(* CODESYS project boiler2.project
   Title: testPrj
   Version: 0.0.0.0

Project tree, tasks and I/O mapping:
  MyController : TM241CE40R, Schneider Electric, order no. TM241CE40R, version 4.0.2.20
    application Application
      libraries: Toolbox, 2.1.0.0 (Schneider Electric); Util, 3.5.1.0 (System)
      task MAST (freewheeling, priority 15, watchdog 100 ms x 1) calls main, pid_control, XT_output
      task Dempf (cyclic, interval t#50ms, priority 1) calls Analog
      function HiddenPOU [ST]
      global variables GVL
      Prog/
        program main [ST]
        program Analog [FBD]
        program pid_control [FBD]
        program XT_output [ST]
        program SafeTmr [FBD]
    DI : Digital Inputs, Schneider Electric, version 4.0.2.20
        input  idwDI_IDW0 : DWORD  // IDW0
        input  Application.xDrumLH1 : BOOL  // IDW0.I0
        input  Application.xDrumLH2 : BOOL  // IDW0.I1
        input  Application.xDrumLl1 : BOOL  // IDW0.I2
        input  Application.xDrumLl2 : BOOL  // IDW0.I3
        input  Application.xFanRun : BOOL  // IDW0.I4
        input  Application.xExhRun : BOOL  // IDW0.I5
        input  Application.xPumpRun : BOOL  // IDW0.I6
        input  Application.xSafeOn : BOOL  // IDW0.I7
        input  Application.xDrumPh : BOOL  // IDW0.I8
        input  Application.xGasPl : BOOL  // IDW0.I9
        input  Application.xGasPh : BOOL  // IDW0.I10
        input  Application.xAirPl : BOOL  // IDW0.I11
        input  Application.xVacPl : BOOL  // IDW0.I12
        input  Application.xBump : BOOL  // IDW0.I13
        input  Application.xFire1 : BOOL  // IDW0.I14
        input  Application.xTight : BOOL  // IDW0.I15
        input  Application.xStartBn : BOOL  // IDW0.I16
        input  Application.xStopBn : BOOL  // IDW0.I17
        input  Application.xAlarmBn : BOOL  // IDW0.I18
        input  Application.xGasAuto : BOOL  // IDW0.I19
        input  Application.xTermAuto : BOOL  // IDW0.I20
        input  Application.xPumpAuto : BOOL  // IDW0.I21
        input  Application.xExhAuto : BOOL  // IDW0.I22
        input  Application.xFanAuto : BOOL  // IDW0.I23
        input  ibDI_IB1 : BYTE  // IB1
    DQ : Digital Outputs, Schneider Electric, version 4.0.2.20
        output Application.yTermOpen : BOOL  // QW0.Q0
        output Application.yTermClose : BOOL  // QW0.Q1
        output Application.ySuppOpen : BOOL  // QW0.Q2
        output Application.ySuppClose : BOOL  // QW0.Q3
        output Application.yCutofVal : BOOL  // QW0.Q4
        output Application.yBurnerVal : BOOL  // QW0.Q5
        output Application.ySafeVal : BOOL  // QW0.Q6
        output Application.yLitherVal : BOOL  // QW0.Q7
        output Application.yFanStart : BOOL  // QW0.Q8
        output Application.yPumpStart : BOOL  // QW0.Q9
        output Application.yGasOpen : BOOL  // QW0.Q10
        output Application.yGasClose : BOOL  // QW0.Q11
        output Application.yPlcStop : BOOL  // QW0.Q12
        output Application.ySerena : BOOL  // QW0.Q13
        output Application.yLamp : BOOL  // QW0.Q14
        output Application.yIgniter : BOOL  // QW0.Q15
        output qbDQ_QB1 : BYTE  // QB1
        unmapped channels: QW0
    Counters : Counters, Schneider Electric, version 4.0.2.20
    Pulse_Generators : Pulse Generators, Schneider Electric, version 4.0.2.20
    Cartridge_1 : Cartridge, Schneider Electric, version 4.0.2.20
    Cartridge_2 : Cartridge, Schneider Electric, version 4.0.2.20
    IO_Bus : IO bus - TM3, Schneider Electric, version 4.0.2.20
      Module_1 : TM3AQ4/G, Schneider Electric, order no. TM3AQ4/G, version 1.0.0.10
          settings: KPI Configuration.KPI Configuration[0] = 19; KPI Configuration.KPI Configuration[1] = 19; KPI Configuration.KPI Configuration[2] = 19; KPI Configuration.KPI Configuration[3] = 19; KPI Configuration.KPI Configuration[5] = 0; KPI Configuration.KPI Configuration[7] = 0; KPI Configuration.KPI Configuration[9] = 0; KPI Configuration.KPI Configuration[11] = 0; KPI Configuration.KPI Configuration[12] = 160; KPI Configuration.KPI Configuration[13] = 15; KPI Configuration.KPI Configuration[14] = 160; KPI Configuration.KPI Configuration[15] = 15; KPI Configuration.KPI Configuration[16] = 160; KPI Configuration.KPI Configuration[17] = 15; KPI Configuration.KPI Configuration[18] = 160; KPI Configuration.KPI Configuration[19] = 15
          output C0001 : INT  // QW0
          output C0002 : INT  // QW1
          output C0003 : INT  // QW2
          output C0004 : INT  // QW3
          input  ibModule_1_IBStatusQW0 : BYTE  // IBStatusQW0
          input  ibModule_1_IBStatusQW1 : BYTE  // IBStatusQW1
          input  ibModule_1_IBStatusQW2 : BYTE  // IBStatusQW2
          input  ibModule_1_IBStatusQW3 : BYTE  // IBStatusQW3
      Module_2 : TM3AI8/G, Schneider Electric, order no. TM3AI8/G, version 1.0.0.12
          settings: KPI Configuration.KPI Configuration[0] = 35; KPI Configuration.KPI Configuration[1] = 35; KPI Configuration.KPI Configuration[2] = 35; KPI Configuration.KPI Configuration[3] = 35; KPI Configuration.KPI Configuration[4] = 35; KPI Configuration.KPI Configuration[5] = 35; KPI Configuration.KPI Configuration[6] = 35; KPI Configuration.KPI Configuration[7] = 35; KPI Configuration.KPI Configuration[9] = 0; KPI Configuration.KPI Configuration[11] = 0; KPI Configuration.KPI Configuration[13] = 0; KPI Configuration.KPI Configuration[15] = 0; KPI Configuration.KPI Configuration[17] = 0; KPI Configuration.KPI Configuration[19] = 0; KPI Configuration.KPI Configuration[21] = 0; KPI Configuration.KPI Configuration[23] = 0; KPI Configuration.KPI Configuration[24] = 160; KPI Configuration.KPI Configuration[25] = 15; KPI Configuration.KPI Configuration[26] = 160; KPI Configuration.KPI Configuration[27] = 15; KPI Configuration.KPI Configuration[28] = 160; KPI Configuration.KPI Configuration[29] = 15; KPI Configuration.KPI Configuration[30] = 160; KPI Configuration.KPI Configuration[31] = 15; KPI Configuration.KPI Configuration[32] = 160; KPI Configuration.KPI Configuration[33] = 15; KPI Configuration.KPI Configuration[34] = 160; KPI Configuration.KPI Configuration[35] = 15; KPI Configuration.KPI Configuration[36] = 160; KPI Configuration.KPI Configuration[37] = 15; KPI Configuration.KPI Configuration[38] = 160; KPI Configuration.KPI Configuration[39] = 15
          input  A0000 : INT  // IW0
          input  A0001 : INT  // IW1
          input  A0002 : INT  // IW2
          input  A0003 : INT  // IW3
          input  A0004 : INT  // IW4
          input  A0005 : INT  // IW5
          input  A0006 : INT  // IW6
          input  A0007 : INT  // IW7
          input  ibModule_2_IBStatusIW0 : BYTE  // IBStatusIW0
          input  ibModule_2_IBStatusIW1 : BYTE  // IBStatusIW1
          input  ibModule_2_IBStatusIW2 : BYTE  // IBStatusIW2
          input  ibModule_2_IBStatusIW3 : BYTE  // IBStatusIW3
          input  ibModule_2_IBStatusIW4 : BYTE  // IBStatusIW4
          input  ibModule_2_IBStatusIW5 : BYTE  // IBStatusIW5
          input  ibModule_2_IBStatusIW6 : BYTE  // IBStatusIW6
          input  ibModule_2_IBStatusIW7 : BYTE  // IBStatusIW7
      Module_3 : TM3AI8/G, Schneider Electric, order no. TM3AI8/G, version 1.0.0.12
          settings: KPI Configuration.KPI Configuration[0] = 35; KPI Configuration.KPI Configuration[1] = 35; KPI Configuration.KPI Configuration[2] = 35; KPI Configuration.KPI Configuration[3] = 35; KPI Configuration.KPI Configuration[4] = 35; KPI Configuration.KPI Configuration[5] = 35; KPI Configuration.KPI Configuration[6] = 35; KPI Configuration.KPI Configuration[7] = 35; KPI Configuration.KPI Configuration[9] = 0; KPI Configuration.KPI Configuration[11] = 0; KPI Configuration.KPI Configuration[13] = 0; KPI Configuration.KPI Configuration[15] = 0; KPI Configuration.KPI Configuration[17] = 0; KPI Configuration.KPI Configuration[19] = 0; KPI Configuration.KPI Configuration[21] = 0; KPI Configuration.KPI Configuration[23] = 0; KPI Configuration.KPI Configuration[24] = 160; KPI Configuration.KPI Configuration[25] = 15; KPI Configuration.KPI Configuration[26] = 160; KPI Configuration.KPI Configuration[27] = 15; KPI Configuration.KPI Configuration[28] = 160; KPI Configuration.KPI Configuration[29] = 15; KPI Configuration.KPI Configuration[30] = 160; KPI Configuration.KPI Configuration[31] = 15; KPI Configuration.KPI Configuration[32] = 160; KPI Configuration.KPI Configuration[33] = 15; KPI Configuration.KPI Configuration[34] = 160; KPI Configuration.KPI Configuration[35] = 15; KPI Configuration.KPI Configuration[36] = 232; KPI Configuration.KPI Configuration[37] = 3; KPI Configuration.KPI Configuration[38] = 160; KPI Configuration.KPI Configuration[39] = 15
          input  A0010 : INT  // IW0
          input  A0011 : INT  // IW1
          input  A0012 : INT  // IW2
          input  A0013 : INT  // IW3
          input  A0014 : INT  // IW4
          input  A0015 : INT  // IW5
          input  A0016 : INT  // IW6
          input  A0017 : INT  // IW7
          input  ibModule_3_IBStatusIW0 : BYTE  // IBStatusIW0
          input  ibModule_3_IBStatusIW1 : BYTE  // IBStatusIW1
          input  ibModule_3_IBStatusIW2 : BYTE  // IBStatusIW2
          input  ibModule_3_IBStatusIW3 : BYTE  // IBStatusIW3
          input  ibModule_3_IBStatusIW4 : BYTE  // IBStatusIW4
          input  ibModule_3_IBStatusIW5 : BYTE  // IBStatusIW5
          input  ibModule_3_IBStatusIW6 : BYTE  // IBStatusIW6
          input  ibModule_3_IBStatusIW7 : BYTE  // IBStatusIW7
      Module_4 : TM3AI8/G, Schneider Electric, order no. TM3AI8/G, version 1.0.0.12
          settings: KPI Configuration.KPI Configuration[0] = 35; KPI Configuration.KPI Configuration[1] = 35; KPI Configuration.KPI Configuration[2] = 35; KPI Configuration.KPI Configuration[3] = 35; KPI Configuration.KPI Configuration[4] = 35; KPI Configuration.KPI Configuration[5] = 35; KPI Configuration.KPI Configuration[6] = 35; KPI Configuration.KPI Configuration[7] = 35; KPI Configuration.KPI Configuration[9] = 0; KPI Configuration.KPI Configuration[11] = 0; KPI Configuration.KPI Configuration[13] = 0; KPI Configuration.KPI Configuration[15] = 0; KPI Configuration.KPI Configuration[17] = 0; KPI Configuration.KPI Configuration[19] = 0; KPI Configuration.KPI Configuration[21] = 0; KPI Configuration.KPI Configuration[23] = 0; KPI Configuration.KPI Configuration[24] = 160; KPI Configuration.KPI Configuration[25] = 15; KPI Configuration.KPI Configuration[26] = 160; KPI Configuration.KPI Configuration[27] = 15; KPI Configuration.KPI Configuration[28] = 160; KPI Configuration.KPI Configuration[29] = 15; KPI Configuration.KPI Configuration[30] = 160; KPI Configuration.KPI Configuration[31] = 15; KPI Configuration.KPI Configuration[32] = 160; KPI Configuration.KPI Configuration[33] = 15; KPI Configuration.KPI Configuration[34] = 160; KPI Configuration.KPI Configuration[35] = 15; KPI Configuration.KPI Configuration[36] = 160; KPI Configuration.KPI Configuration[37] = 15; KPI Configuration.KPI Configuration[38] = 160; KPI Configuration.KPI Configuration[39] = 15
          input  A0020 : INT  // IW0
          input  A0021 : INT  // IW1
          input  A0022 : INT  // IW2
          input  A0023 : INT  // IW3
          input  A0024 : INT  // IW4
          input  A0025 : INT  // IW5
          input  A0026 : INT  // IW6
          input  A0027 : INT  // IW7
          input  ibModule_4_IBStatusIW0 : BYTE  // IBStatusIW0
          input  ibModule_4_IBStatusIW1 : BYTE  // IBStatusIW1
          input  ibModule_4_IBStatusIW2 : BYTE  // IBStatusIW2
          input  ibModule_4_IBStatusIW3 : BYTE  // IBStatusIW3
          input  ibModule_4_IBStatusIW4 : BYTE  // IBStatusIW4
          input  ibModule_4_IBStatusIW5 : BYTE  // IBStatusIW5
          input  ibModule_4_IBStatusIW6 : BYTE  // IBStatusIW6
          input  ibModule_4_IBStatusIW7 : BYTE  // IBStatusIW7
    COM_Bus : COM bus, Schneider Electric, version 4.0.2.20
    Ethernet_1 : Ethernet Network, Schneider Electric, version 4.0.2.20
        settings: IPAddress = [192, 168, 15, 152]; SubnetMask = [255, 255, 255, 0]; GatewayAddress = [192, 168, 15, 1]; DeviceName = 'boiler2'; WebServer = FALSE; FTP Server = FALSE; SoMachine Protocol = TRUE; Modbus Server = TRUE; NetManage Protocol = FALSE; SNMP protocol = FALSE; Enable Routing = FALSE; WebVisu protocol = FALSE
      ModbusTCP_Slave_Device : ModbusTCP Slave Device, Schneider Electric, version 3.5.2.3
          unmapped channels: Inputs, Outputs
    Serial_Line_1 : Serial line, Schneider Electric, version 4.0.2.20
    Serial_Line_2 : Serial line, Schneider Electric, version 4.0.2.20
      Modbus_IOScanner : Modbus IOScanner, Schneider Electric, version 3.5.3.6
        Generic_Modbus_Slave : Generic Modbus Slave, Schneider Electric, version 3.5.3.6
            settings: Channel 1.Function Code = 3; Channel 1.Read Offset = 16#1001; Channel 1.Read Length = 6; Channel 1.Write Offset = 0; Channel 1.Write Length = 0; Channel 1.Cycle Time = 100; Channel 2.Function Code = 3; Channel 2.Read Offset = 16#8000; Channel 2.Read Length = 1; Channel 2.Write Offset = 0; Channel 2.Write Length = 0; Channel 2.Cycle Time = 100; Channel 3.Function Code = 3; Channel 3.Read Offset = 16#3000; Channel 3.Read Length = 1; Channel 3.Write Offset = 0; Channel 3.Write Length = 0; Channel 3.Cycle Time = 100
            input  M1 : WORD  // Channel 1.Channel 1[0]
            input  M2 : WORD  // Channel 1.Channel 1[1]
            input  M3 : WORD  // Channel 1.Channel 1[2]
            input  M4 : WORD  // Channel 1.Channel 1[3]
            input  M5 : WORD  // Channel 1.Channel 1[4]
            input  M6 : WORD  // Channel 1.Channel 1[5]
            input  M7 : WORD  // Channel 2.Channel 2[0]
            input  M8 : WORD  // Channel 3.Channel 3[0]
            unmapped channels: Channel 1, Channel 2, Channel 3
*)

// MyController/Application/GVL
VAR_GLOBAL

// run
	Run AT %M9: BOOL;
// DI
xDrumLH1 AT %M10: BOOL;
xDrumLH2 AT %M11: BOOL;
xDrumLl1 AT %M12: BOOL;
xDrumLl2 AT %M13: BOOL;
xFanRun AT %M14: BOOL;
xExhRun AT %M15: BOOL;
xPumpRun AT %M16: BOOL;
xSafeOn AT %M17: BOOL;
xDrumPh AT %M18: BOOL;
xGasPl AT %M19: BOOL;
xGasPh AT %M20: BOOL;
xAirPl AT %M21: BOOL;
xVacPl AT %M22: BOOL;
xBump AT %M23: BOOL;
xFire1 AT %M24: BOOL;
xTight AT %M25: BOOL;
xStartBn AT %M26: BOOL;
xStopBn AT %M27: BOOL;
xAlarmBn AT %M28: BOOL;
xGasAuto AT %M29: BOOL;
xTermAuto AT %M30: BOOL;
xPumpAuto AT %M31: BOOL;
xExhAuto AT %M32: BOOL;
xFanAuto AT %M33: BOOL;
// DO
yCutofVal AT %M34: BOOL;
yBurnerVal AT %M35: BOOL;
ySafeVal AT %M36: BOOL;
yLitherVal AT %M37: BOOL;
yIgniter AT %M38: BOOL;
yFanStart AT %M39: BOOL;
yPumpStart AT %M40: BOOL;
yGasOpen AT %M41: BOOL;
yGasClose AT %M42: BOOL;
yTermOpen AT %M43: BOOL;
yTermClose AT %M44: BOOL;
ySuppOpen AT %M45: BOOL;
ySuppClose AT %M46: BOOL;
yPlcStop AT %M47: BOOL;
ySerena AT %M48: BOOL;
yLamp AT %M49: BOOL;
//прапори аварійних сигналів
Alm0001 AT %M50: BOOL;
Alm0002 AT %M51: BOOL;
Alm0003 AT %M52: BOOL;
Alm0004 AT %M53: BOOL;
Alm0005 AT %M54: BOOL;
Alm0006 AT %M55: BOOL;
Alm0007 AT %M56: BOOL;
Alm0008 AT %M57: BOOL;
Alm0009 AT %M58: BOOL;
Alm0010 AT %M59: BOOL;
Alm0011 AT %M60: BOOL;
Alm0012 AT %M61: BOOL;
alFire1 AT %M62: BOOL;
alFan AT %M63: BOOL;
alExh AT %M64: BOOL;
alPump AT %M65: BOOL;
alSupport AT %M66: BOOL;

Alert AT %M123: BOOL;
Halt AT %M124: BOOL;
prLock AT %M125: BOOL;
Cvit AT %M126: BOOL;


amGas AT %M100: BOOL;
amTerm AT %M101: BOOL;
amSupport AT %M102: BOOL;
AM0001 AT %M103: BOOL;
AM0002 AT %M104: BOOL;
AM0003 AT %M105: BOOL;
AM0004 AT %M106: BOOL;
AM0005 AT %M107: BOOL;
AM0006 AT %M108: BOOL;



Fgas AT %MD9: REAL;
Fpara AT %MD10: REAL;
Fwater AT %MD11: REAL;
Fair AT %MD12: REAL;
Ldrum AT %MD13: REAL;
Pg15a AT %MD14: REAL;
Ppara AT %MD15: REAL;
Pp7a AT %MD16: REAL;

Tpar AT %MD17: REAL;
Tv3a AT %MD18: REAL;
Tv4a AT %MD19: REAL;
Tk AT %MD20: REAL;
Ta5a AT %MD21: REAL;
Ta6a AT %MD22: REAL;
Tp17a AT %MD23: REAL;
Tp18a AT %MD24: REAL;

Pair AT %MD25: REAL;
Pvac AT %MD26: REAL;
Pv12a AT %MD27: REAL;
gGas AT %MD28: REAL;
gTerm AT %MD49: REAL;
gSupp AT %MD51: REAL;
QO2fume AT %MD53: REAL;
Vx AT %MD55: REAL;

cPump AT %MD57: REAL;
cFan AT %MD59: REAL;
cExh AT %MD61: REAL;
cGas AT %MD63: REAL;
cTerm AT %MD65: REAL;
cSupport AT %MD67: REAL;
cX AT %MD69: REAL;


fA0000 AT %MW100: UINT;
fA0001 AT %MW101: UINT;
fA0002 AT %MW102: UINT;
fA0003 AT %MW103: UINT;
fA0004 AT %MW104: UINT;
fA0005 AT %MW105: UINT;
fA0006 AT %MW106: UINT;
fA0007 AT %MW107: UINT;
fA0010 AT %MW108: UINT;
fA0011 AT %MW109: UINT;
fA0012 AT %MW110: UINT;
fA0013 AT %MW111: UINT;
fA0014 AT %MW112: UINT;
fA0015 AT %MW113: UINT;
fA0016 AT %MW114: UINT;
fA0017 AT %MW115: UINT;
fA0020 AT %MW116: UINT;
fA0021 AT %MW117: UINT;
fA0022 AT %MW118: UINT;
fA0023 AT %MW119: UINT;
fA0024 AT %MW120: UINT;
fA0025 AT %MW121: UINT;
fA0026 AT %MW122: UINT;
fA0027 AT %MW123: UINT;

dGas AT %MD124: REAL;
dTerm AT %MD126: REAL;
dSupport AT %MD127: REAL;

Sp0001 AT %MD377: REAL;
Kp0001 AT %MD379: REAL;
Ti0001 AT %MD381: REAL;
Td0001 AT %MD383: REAL;
Xmin0001 AT %MD385: REAL;
Xmax0001 AT %MD387: REAL;

Sp0002 AT %MD389: REAL;
Kp0002 AT %MD391: REAL;
Ti0002 AT %MD393: REAL;
Td0002 AT %MD395: REAL;
Xmin0002 AT %MD397: REAL;
Xmax0002 AT %MD399: REAL;

Sp0003 AT %MD401: REAL;
Kp0003 AT %MD403: REAL;
Ti0003 AT %MD405: REAL;
Td0003 AT %MD407: REAL;
Xmin0003 AT %MD409: REAL;
Xmax0003 AT %MD411: REAL;

Sp0004 AT %MD413: REAL;
Kp0004 AT %MD415: REAL;
Ti0004 AT %MD417: REAL;
Td0004 AT %MD419: REAL;
Xmin0004 AT %MD421: REAL;
Xmax0004 AT %MD423: REAL;

Sp0005 AT %MD425: REAL;
Kp0005 AT %MD427: REAL;
Ti0005 AT %MD429: REAL;
Td0005 AT %MD431: REAL;
Xmin0005 AT %MD433: REAL;
Xmax0005 AT %MD435: REAL;

Sp0006 AT %MD437: REAL;
Kp0006 AT %MD439: REAL;
Ti0006 AT %MD441: REAL;
Td0006 AT %MD443: REAL;
Xmin0006 AT %MD445: REAL;
Xmax0006 AT %MD447: REAL;
// таймери аварій мео
tMeoTerm AT %MD449: REAL;
tMeoGas AT %MD451: REAL;

// таймери аварійних сигналізацій
Tpr0001 AT %ML511: TIME;
Tpr0002 AT %ML513: TIME;
Tpr0003 AT %ML515: TIME;
Tpr0004 AT %ML517: TIME;
Tpr0005 AT %ML519: TIME;
Tpr0006 AT %ML521: TIME;
Tpr0007 AT %ML523: TIME;
Tpr0008 AT %ML525: TIME;
Tpr0009 AT %ML527: TIME;
Tpr0010 AT %ML529: TIME;
Tpr0011 AT %ML531: TIME;
Tpr0012 AT %ML533: TIME;

	Xt0001: REAL;
	Xt0002: REAL;
	Xt0003: REAL;
	Xt0004: REAL;
	Xt0005: REAL;
	Xt0006: REAL;
	
	tMeo1: TIME;
	tMeo2: TIME;
	tMeo3: TIME;

END_VAR

// MyController/Application/Prog/main
PROGRAM main
VAR
	fe_amGas: F_TRIG;
	fe_amTerm: F_TRIG;
	fe_amSupport: F_TRIG;
END_VAR

(*Робота з МЕО*)
(*Газ*)
(*Взагалі-то вся ця хрінь проситься зробити блоком але як тоді в ручну управляти виходами ? треба подумати*)
IF amGas OR AM0004 THEN
	IF gGas>cGas+dGas THEN (*якщо відкрито більше ніж треба*)
		IF NOT yGasClose THEN (*В перший момент розрахувати значення таймера на виконання операції*) 
			tMeo1:=REAL_TO_TIME(ABS(gGas-cGas)*tMeoGas);
		END_IF;		
		yGasClose:=TRUE; (*відкрити*)
	END_IF;
	IF gGas<cGas-dGas THEN (*як закрито більше ніж треба*)
		IF NOT yGasOpen THEN 
			tMeo1:=REAL_TO_TIME(ABS(gGas-cGas)*tMeoGas);
		END_IF;		
		yGasOpen:=TRUE;
	END_IF;
	IF gGas<cGas THEN
		yGasClose:=FALSE;
	END_IF;
	IF gGas>cGas THEN 
		yGasOpen:=FALSE;
	END_IF;
END_IF;

(*при переході в ручний режим виключити виходи, якщов включені*)
fe_amGas(CLK:=amGas);
IF fe_amGas.Q THEN
	yGasOpen:=FALSE;
	yGasClose:=FALSE;
END_IF;


(*Температура*)
IF amTerm OR AM0005 THEN
	IF gTerm>cTerm+dTerm THEN (*якщо відкрито більге ніж треба*)
		IF NOT yTermClose THEN
			tMeo2:=REAL_TO_TIME(ABS(gTerm-cTerm)*tMeoTerm);		
		END_IF;
		yTermClose:=TRUE; (*відкрити*)
	END_IF;
	IF gTerm<cTerm-dTerm THEN (*як закрито більше ніж треба*)
		IF NOT yTermOpen THEN
			tMeo2:=REAL_TO_TIME(ABS(gTerm-cTerm)*tMeoTerm);		
		END_IF;
		tMeo2:=REAL_TO_TIME(ABS(gTerm-cTerm)*tMeoTerm);
		yTermOpen:=TRUE;
	END_IF;
	IF gTerm<cTerm THEN
		yTermClose:=FALSE;
	END_IF;
	IF gTerm>cTerm THEN 
		yTermOpen:=FALSE;
	END_IF;
END_IF;

(*при переході в ручний режим виключити виходи, якщов включені*)
fe_amTerm(CLK:=amTerm);
IF fe_amTerm.Q THEN
	yTermOpen:=FALSE;
	yTermClose:=FALSE;
END_IF;

(*підпір*)
IF amSupport OR AM0005  THEN
	cSupport:=4000.0-cTerm; (*клапан підпору працює в противофазі із клапаном температури*)
	IF gSupp>cSupport+dSupport THEN (*якщо відкрито більге ніж треба*)
		IF NOT ySuppClose THEN
			tMeo3:=REAL_TO_TIME(ABS(gSupp-cSupport)*tMeoTerm);				
		END_IF;
		ySuppClose:=TRUE; (*відкрити*)
	END_IF;
	IF gSupp<cSupport-dSupport THEN (*як закрито більше ніж треба*)
		IF NOT ySuppOpen THEN
			tMeo3:=REAL_TO_TIME(ABS(gSupp-cSupport)*tMeoTerm);		
		END_IF;
		ySuppOpen:=TRUE;
	END_IF;
	IF gSupp<cSupport THEN
		ySuppClose:=FALSE;
	END_IF;
	IF gSupp>cSupport THEN 
		ySuppOpen:=FALSE;
	END_IF;
END_IF;

(*при переході в ручний режим виключити виходи, якщов включені*)
fe_amSupport(CLK:=amSupport);
IF fe_amSupport.Q THEN
	ySuppOpen:=FALSE;
	ySuppClose:=FALSE;
END_IF;
(*----------------------------------------------------------------------------------------------------------------------------------*)

END_PROGRAM

// MyController/Application/Prog/pid_control
PROGRAM pid_control
VAR
	pid1: Util.PID;
	pid2: Util.PID;
	pid3: Util.PID;
	pid4: Util.PID;
	pid5: Util.PID;
	pid6: Util.PID;
END_VAR
VAR // added by the converter: edge detectors and wires of the graphical bodies
    _rt1, _rt2, _rt3, _rt4, _rt5, _rt6 : R_TRIG;
END_VAR

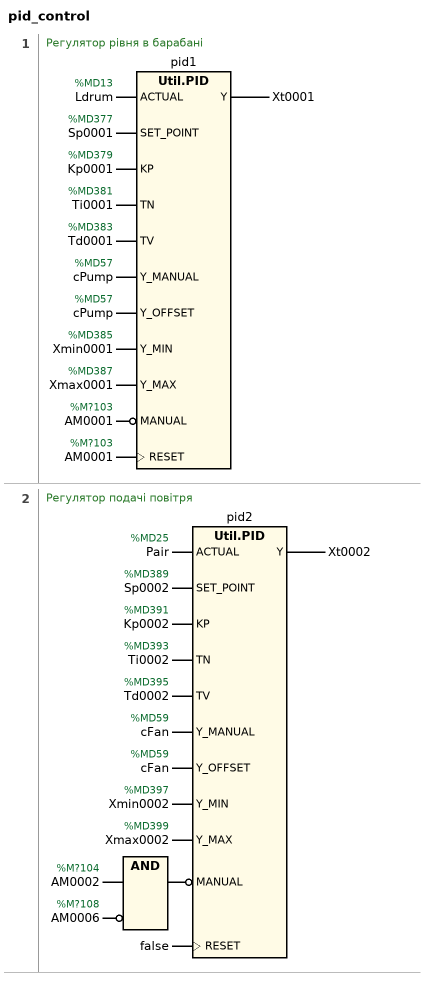
// NETWORK 1
// Регулятор рівня в барабані
//   Ldrum: AT %MD13
//   Sp0001: AT %MD377
//   Kp0001: AT %MD379
//   Ti0001: AT %MD381
//   Td0001: AT %MD383
//   cPump: AT %MD57
//   Xmin0001: AT %MD385
//   Xmax0001: AT %MD387
//   AM0001: AT %M?103
_rt1(CLK := AM0001);
pid1(
    ACTUAL := Ldrum,
    SET_POINT := Sp0001,
    KP := Kp0001,
    TN := Ti0001,
    TV := Td0001,
    Y_MANUAL := cPump,
    Y_OFFSET := cPump,
    Y_MIN := Xmin0001,
    Y_MAX := Xmax0001,
    MANUAL := NOT AM0001,
    RESET := _rt1.Q); // Util.PID
Xt0001 := pid1.Y;

// NETWORK 2
// Регулятор подачі повітря
//   Pair: AT %MD25
//   Sp0002: AT %MD389
//   Kp0002: AT %MD391
//   Ti0002: AT %MD393
//   Td0002: AT %MD395
//   cFan: AT %MD59
//   Xmin0002: AT %MD397
//   Xmax0002: AT %MD399
//   AM0002: AT %M?104
//   AM0006: AT %M?108
_rt2(CLK := false);
pid2(
    ACTUAL := Pair,
    SET_POINT := Sp0002,
    KP := Kp0002,
    TN := Ti0002,
    TV := Td0002,
    Y_MANUAL := cFan,
    Y_OFFSET := cFan,
    Y_MIN := Xmin0002,
    Y_MAX := Xmax0002,
    MANUAL := NOT (AM0002 AND NOT AM0006),
    RESET := _rt2.Q); // Util.PID
Xt0002 := pid2.Y;

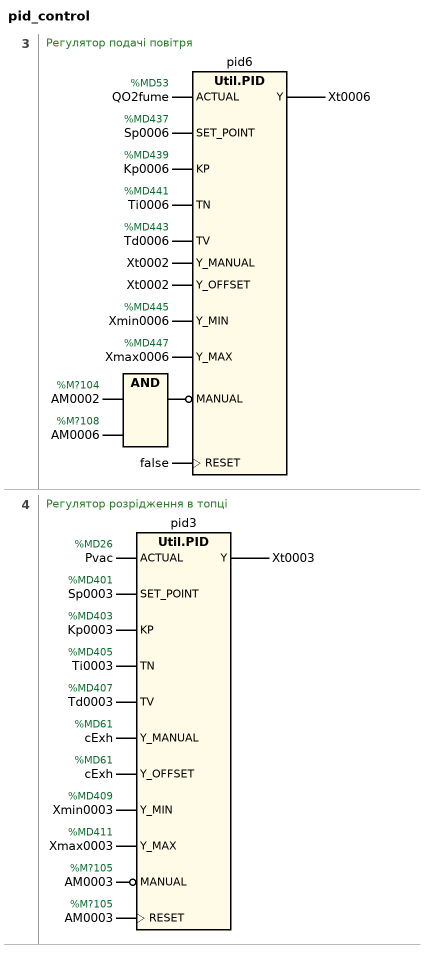
// NETWORK 3
// Регулятор подачі повітря
//   QO2fume: AT %MD53
//   Sp0006: AT %MD437
//   Kp0006: AT %MD439
//   Ti0006: AT %MD441
//   Td0006: AT %MD443
//   Xmin0006: AT %MD445
//   Xmax0006: AT %MD447
//   AM0002: AT %M?104
//   AM0006: AT %M?108
_rt3(CLK := false);
pid6(
    ACTUAL := QO2fume,
    SET_POINT := Sp0006,
    KP := Kp0006,
    TN := Ti0006,
    TV := Td0006,
    Y_MANUAL := Xt0002,
    Y_OFFSET := Xt0002,
    Y_MIN := Xmin0006,
    Y_MAX := Xmax0006,
    MANUAL := NOT (AM0002 AND AM0006),
    RESET := _rt3.Q); // Util.PID
Xt0006 := pid6.Y;

// NETWORK 4
// Регулятор розрідження в топці
//   Pvac: AT %MD26
//   Sp0003: AT %MD401
//   Kp0003: AT %MD403
//   Ti0003: AT %MD405
//   Td0003: AT %MD407
//   cExh: AT %MD61
//   Xmin0003: AT %MD409
//   Xmax0003: AT %MD411
//   AM0003: AT %M?105
_rt4(CLK := AM0003);
pid3(
    ACTUAL := Pvac,
    SET_POINT := Sp0003,
    KP := Kp0003,
    TN := Ti0003,
    TV := Td0003,
    Y_MANUAL := cExh,
    Y_OFFSET := cExh,
    Y_MIN := Xmin0003,
    Y_MAX := Xmax0003,
    MANUAL := NOT AM0003,
    RESET := _rt4.Q); // Util.PID
Xt0003 := pid3.Y;

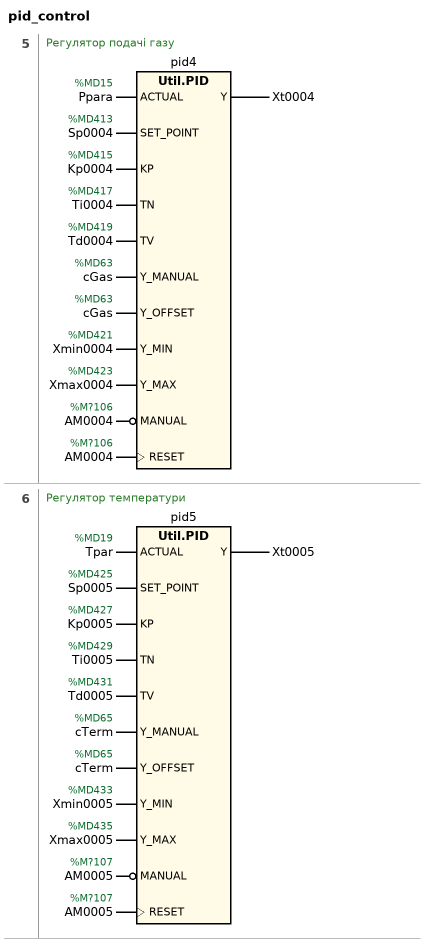
// NETWORK 5
// Регулятор подачі газу
//   Ppara: AT %MD15
//   Sp0004: AT %MD413
//   Kp0004: AT %MD415
//   Ti0004: AT %MD417
//   Td0004: AT %MD419
//   cGas: AT %MD63
//   Xmin0004: AT %MD421
//   Xmax0004: AT %MD423
//   AM0004: AT %M?106
_rt5(CLK := AM0004);
pid4(
    ACTUAL := Ppara,
    SET_POINT := Sp0004,
    KP := Kp0004,
    TN := Ti0004,
    TV := Td0004,
    Y_MANUAL := cGas,
    Y_OFFSET := cGas,
    Y_MIN := Xmin0004,
    Y_MAX := Xmax0004,
    MANUAL := NOT AM0004,
    RESET := _rt5.Q); // Util.PID
Xt0004 := pid4.Y;

// NETWORK 6
// Регулятор температури
//   Tpar: AT %MD19
//   Sp0005: AT %MD425
//   Kp0005: AT %MD427
//   Ti0005: AT %MD429
//   Td0005: AT %MD431
//   cTerm: AT %MD65
//   Xmin0005: AT %MD433
//   Xmax0005: AT %MD435
//   AM0005: AT %M?107
_rt6(CLK := AM0005);
pid5(
    ACTUAL := Tpar,
    SET_POINT := Sp0005,
    KP := Kp0005,
    TN := Ti0005,
    TV := Td0005,
    Y_MANUAL := cTerm,
    Y_OFFSET := cTerm,
    Y_MIN := Xmin0005,
    Y_MAX := Xmax0005,
    MANUAL := NOT AM0005,
    RESET := _rt6.Q); // Util.PID
Xt0005 := pid5.Y;

END_PROGRAM

// MyController/Application/Prog/XT_output
PROGRAM XT_output
VAR
	fe_am0001: F_TRIG;
	fe_am0002: F_TRIG;
	fe_am0003: F_TRIG;
	fe_am0004: F_TRIG;
	fe_am0005: F_TRIG;

	re_am0001: R_TRIG;
	re_am0002: R_TRIG;
	re_am0003: R_TRIG;
	re_am0004: R_TRIG;
	re_am0005: R_TRIG;

END_VAR

IF Am0001 THEN
	cPump:=Xt0001;
END_IF;

IF Am0002 THEN
	cFan:=Xt0006;
END_IF;

IF Am0003 THEN
	cExh:=Xt0003;
END_IF;

IF Am0004 THEN
	cGas:=Xt0004;
END_IF;

IF Am0005 THEN
	cTerm:=Xt0005;
END_IF;

(*Управління перемикачами ручний-автомати*)
re_AM0001(CLK:=xPumpAuto);
fe_AM0001(CLK:=xPumpAuto);

IF re_AM0001.Q THEN
	AM0001:=TRUE;
END_IF;

IF fe_AM0001.Q THEN
	AM0001:=FALSE;
END_IF;
(*-------------------------------------*)
re_AM0002(CLK:=xFanAuto);
fe_AM0002(CLK:=xFanAuto);

IF re_AM0002.Q THEN
	AM0002:=TRUE;
END_IF;

IF fe_AM0002.Q THEN
	AM0002:=FALSE;
END_IF;
(*-------------------------------------*)
re_AM0003(CLK:=xExhAuto);
fe_AM0003(CLK:=xExhAuto);

IF re_AM0003.Q THEN
	AM0003:=TRUE;
END_IF;

IF fe_AM0003.Q THEN
	AM0003:=FALSE;
END_IF;
(*-------------------------------------*)
re_AM0004(CLK:=xGasAuto);
fe_AM0004(CLK:=xGasAuto);

IF re_AM0004.Q THEN
	AM0004:=TRUE;
END_IF;

IF fe_AM0004.Q THEN
	AM0004:=FALSE;
END_IF;
(*-------------------------------------*)
re_AM0005(CLK:=xTermAuto);
fe_AM0005(CLK:=xTermAuto);

IF re_AM0005.Q THEN
	AM0005:=TRUE;
END_IF;

IF fe_AM0005.Q THEN
	AM0005:=FALSE;
END_IF;
(*-------------------------------------*)

END_PROGRAM

// MyController/Application/Prog/Analog
PROGRAM Analog
VAR
avg0000: SE_TBX.Filter_MovingAverage;
avg0001: SE_TBX.Filter_MovingAverage;
avg0002: SE_TBX.Filter_MovingAverage;
avg0003: SE_TBX.Filter_MovingAverage;
avg0004: SE_TBX.Filter_MovingAverage;
avg0005: SE_TBX.Filter_MovingAverage;
avg0006: SE_TBX.Filter_MovingAverage;
avg0007: SE_TBX.Filter_MovingAverage;
avg0010: SE_TBX.Filter_MovingAverage;
avg0011: SE_TBX.Filter_MovingAverage;
avg0012: SE_TBX.Filter_MovingAverage;
avg0013: SE_TBX.Filter_MovingAverage;
avg0014: SE_TBX.Filter_MovingAverage;
avg0015: SE_TBX.Filter_MovingAverage;
avg0016: SE_TBX.Filter_MovingAverage;
avg0017: SE_TBX.Filter_MovingAverage;
avg0020: SE_TBX.Filter_MovingAverage;
avg0021: SE_TBX.Filter_MovingAverage;
avg0022: SE_TBX.Filter_MovingAverage;
avg0023: SE_TBX.Filter_MovingAverage;
avg0024: SE_TBX.Filter_MovingAverage;
avg0025: SE_TBX.Filter_MovingAverage;
avg0026: SE_TBX.Filter_MovingAverage;
avg0027: SE_TBX.Filter_MovingAverage;

END_VAR
VAR
END_VAR
VAR // added by the converter: edge detectors and wires of the graphical bodies
    _rt1, _rt2, _rt3, _rt4, _rt5, _rt6, _rt7, _rt8, _rt9, _rt10, _rt11, _rt12, _rt13, _rt14, _rt15, _rt16, _rt17, _rt18, _rt19, _rt20, _rt21, _rt22, _rt23, _rt24 : R_TRIG;
END_VAR

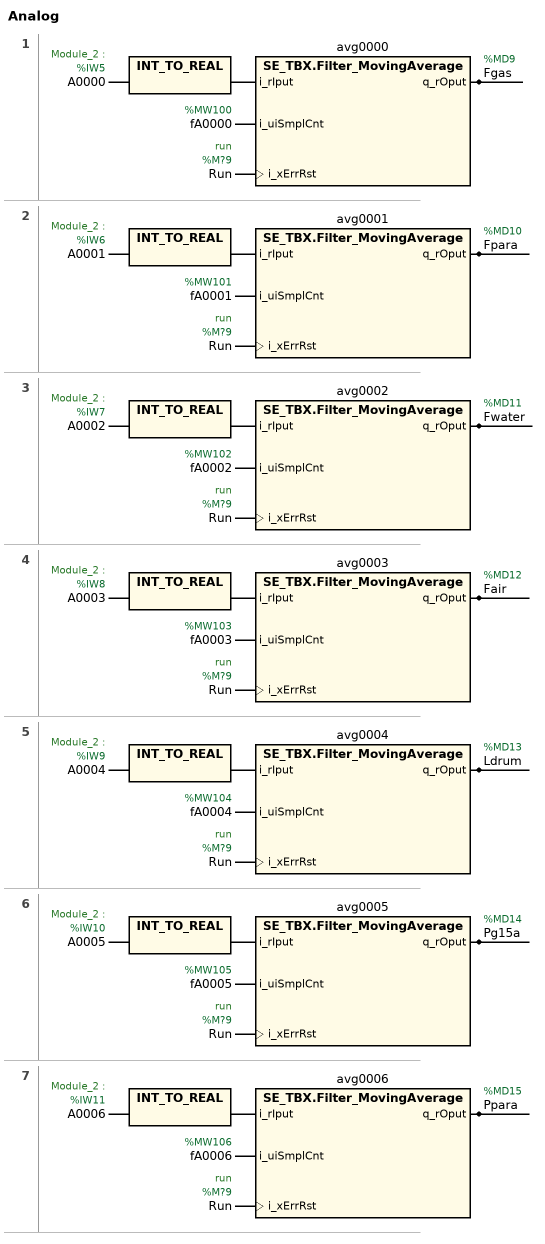
// NETWORK 1
//   A0000: Module_2 : | AT %IW5
//   fA0000: AT %MW100
//   Run: run | AT %M?9
//   Fgas: AT %MD9
_rt1(CLK := Run);
avg0000(i_rIput := INT_TO_REAL(A0000), i_uiSmplCnt := fA0000, i_xErrRst := _rt1.Q, q_rOput => Fgas); // SE_TBX.Filter_MovingAverage

// NETWORK 2
//   A0001: Module_2 : | AT %IW6
//   fA0001: AT %MW101
//   Run: run | AT %M?9
//   Fpara: AT %MD10
_rt2(CLK := Run);
avg0001(i_rIput := INT_TO_REAL(A0001), i_uiSmplCnt := fA0001, i_xErrRst := _rt2.Q, q_rOput => Fpara); // SE_TBX.Filter_MovingAverage

// NETWORK 3
//   A0002: Module_2 : | AT %IW7
//   fA0002: AT %MW102
//   Run: run | AT %M?9
//   Fwater: AT %MD11
_rt3(CLK := Run);
avg0002(i_rIput := INT_TO_REAL(A0002), i_uiSmplCnt := fA0002, i_xErrRst := _rt3.Q, q_rOput => Fwater); // SE_TBX.Filter_MovingAverage

// NETWORK 4
//   A0003: Module_2 : | AT %IW8
//   fA0003: AT %MW103
//   Run: run | AT %M?9
//   Fair: AT %MD12
_rt4(CLK := Run);
avg0003(i_rIput := INT_TO_REAL(A0003), i_uiSmplCnt := fA0003, i_xErrRst := _rt4.Q, q_rOput => Fair); // SE_TBX.Filter_MovingAverage

// NETWORK 5
//   A0004: Module_2 : | AT %IW9
//   fA0004: AT %MW104
//   Run: run | AT %M?9
//   Ldrum: AT %MD13
_rt5(CLK := Run);
avg0004(i_rIput := INT_TO_REAL(A0004), i_uiSmplCnt := fA0004, i_xErrRst := _rt5.Q, q_rOput => Ldrum); // SE_TBX.Filter_MovingAverage

// NETWORK 6
//   A0005: Module_2 : | AT %IW10
//   fA0005: AT %MW105
//   Run: run | AT %M?9
//   Pg15a: AT %MD14
_rt6(CLK := Run);
avg0005(i_rIput := INT_TO_REAL(A0005), i_uiSmplCnt := fA0005, i_xErrRst := _rt6.Q, q_rOput => Pg15a); // SE_TBX.Filter_MovingAverage

// NETWORK 7
//   A0006: Module_2 : | AT %IW11
//   fA0006: AT %MW106
//   Run: run | AT %M?9
//   Ppara: AT %MD15
_rt7(CLK := Run);
avg0006(i_rIput := INT_TO_REAL(A0006), i_uiSmplCnt := fA0006, i_xErrRst := _rt7.Q, q_rOput => Ppara); // SE_TBX.Filter_MovingAverage

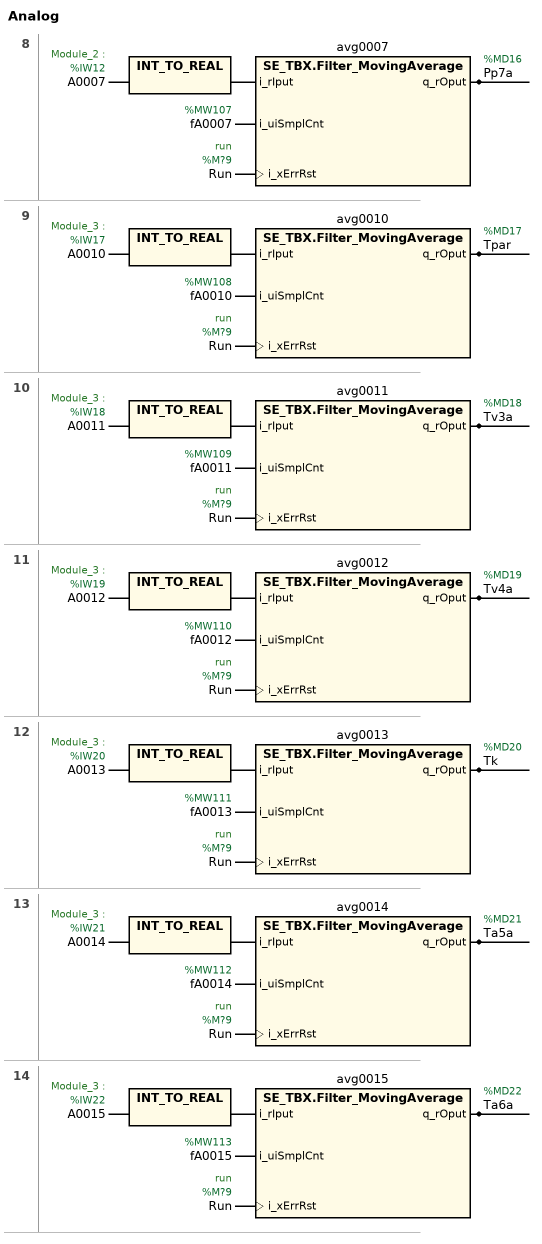
// NETWORK 8
//   A0007: Module_2 : | AT %IW12
//   fA0007: AT %MW107
//   Run: run | AT %M?9
//   Pp7a: AT %MD16
_rt8(CLK := Run);
avg0007(i_rIput := INT_TO_REAL(A0007), i_uiSmplCnt := fA0007, i_xErrRst := _rt8.Q, q_rOput => Pp7a); // SE_TBX.Filter_MovingAverage

// NETWORK 9
//   A0010: Module_3 : | AT %IW17
//   fA0010: AT %MW108
//   Run: run | AT %M?9
//   Tpar: AT %MD17
_rt9(CLK := Run);
avg0010(i_rIput := INT_TO_REAL(A0010), i_uiSmplCnt := fA0010, i_xErrRst := _rt9.Q, q_rOput => Tpar); // SE_TBX.Filter_MovingAverage

// NETWORK 10
//   A0011: Module_3 : | AT %IW18
//   fA0011: AT %MW109
//   Run: run | AT %M?9
//   Tv3a: AT %MD18
_rt10(CLK := Run);
avg0011(i_rIput := INT_TO_REAL(A0011), i_uiSmplCnt := fA0011, i_xErrRst := _rt10.Q, q_rOput => Tv3a); // SE_TBX.Filter_MovingAverage

// NETWORK 11
//   A0012: Module_3 : | AT %IW19
//   fA0012: AT %MW110
//   Run: run | AT %M?9
//   Tv4a: AT %MD19
_rt11(CLK := Run);
avg0012(i_rIput := INT_TO_REAL(A0012), i_uiSmplCnt := fA0012, i_xErrRst := _rt11.Q, q_rOput => Tv4a); // SE_TBX.Filter_MovingAverage

// NETWORK 12
//   A0013: Module_3 : | AT %IW20
//   fA0013: AT %MW111
//   Run: run | AT %M?9
//   Tk: AT %MD20
_rt12(CLK := Run);
avg0013(i_rIput := INT_TO_REAL(A0013), i_uiSmplCnt := fA0013, i_xErrRst := _rt12.Q, q_rOput => Tk); // SE_TBX.Filter_MovingAverage

// NETWORK 13
//   A0014: Module_3 : | AT %IW21
//   fA0014: AT %MW112
//   Run: run | AT %M?9
//   Ta5a: AT %MD21
_rt13(CLK := Run);
avg0014(i_rIput := INT_TO_REAL(A0014), i_uiSmplCnt := fA0014, i_xErrRst := _rt13.Q, q_rOput => Ta5a); // SE_TBX.Filter_MovingAverage

// NETWORK 14
//   A0015: Module_3 : | AT %IW22
//   fA0015: AT %MW113
//   Run: run | AT %M?9
//   Ta6a: AT %MD22
_rt14(CLK := Run);
avg0015(i_rIput := INT_TO_REAL(A0015), i_uiSmplCnt := fA0015, i_xErrRst := _rt14.Q, q_rOput => Ta6a); // SE_TBX.Filter_MovingAverage

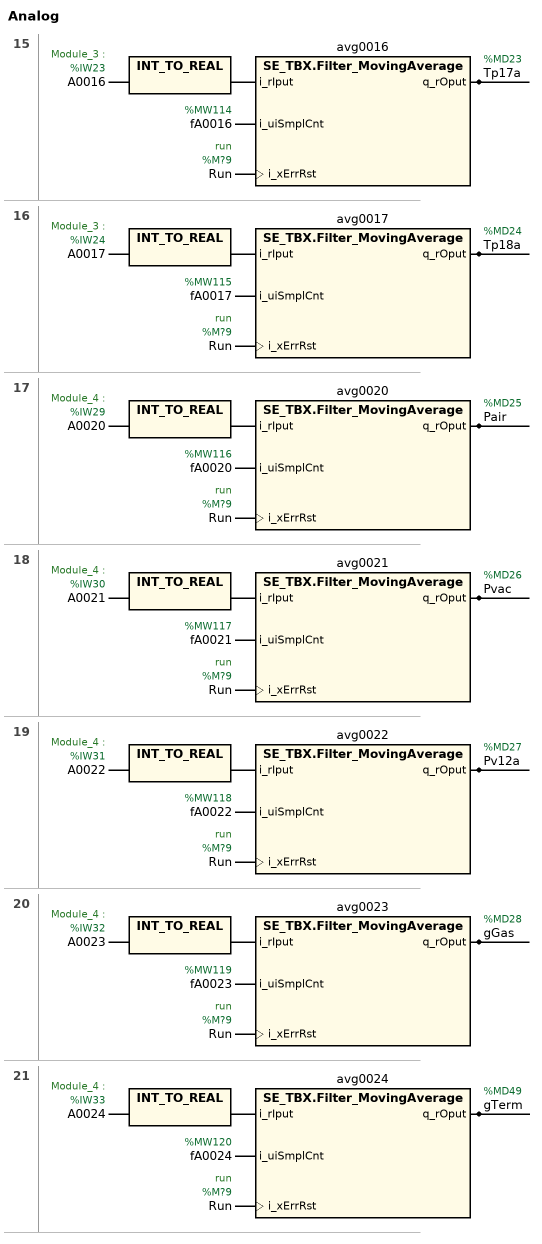
// NETWORK 15
//   A0016: Module_3 : | AT %IW23
//   fA0016: AT %MW114
//   Run: run | AT %M?9
//   Tp17a: AT %MD23
_rt15(CLK := Run);
avg0016(i_rIput := INT_TO_REAL(A0016), i_uiSmplCnt := fA0016, i_xErrRst := _rt15.Q, q_rOput => Tp17a); // SE_TBX.Filter_MovingAverage

// NETWORK 16
//   A0017: Module_3 : | AT %IW24
//   fA0017: AT %MW115
//   Run: run | AT %M?9
//   Tp18a: AT %MD24
_rt16(CLK := Run);
avg0017(i_rIput := INT_TO_REAL(A0017), i_uiSmplCnt := fA0017, i_xErrRst := _rt16.Q, q_rOput => Tp18a); // SE_TBX.Filter_MovingAverage

// NETWORK 17
//   A0020: Module_4 : | AT %IW29
//   fA0020: AT %MW116
//   Run: run | AT %M?9
//   Pair: AT %MD25
_rt17(CLK := Run);
avg0020(i_rIput := INT_TO_REAL(A0020), i_uiSmplCnt := fA0020, i_xErrRst := _rt17.Q, q_rOput => Pair); // SE_TBX.Filter_MovingAverage

// NETWORK 18
//   A0021: Module_4 : | AT %IW30
//   fA0021: AT %MW117
//   Run: run | AT %M?9
//   Pvac: AT %MD26
_rt18(CLK := Run);
avg0021(i_rIput := INT_TO_REAL(A0021), i_uiSmplCnt := fA0021, i_xErrRst := _rt18.Q, q_rOput => Pvac); // SE_TBX.Filter_MovingAverage

// NETWORK 19
//   A0022: Module_4 : | AT %IW31
//   fA0022: AT %MW118
//   Run: run | AT %M?9
//   Pv12a: AT %MD27
_rt19(CLK := Run);
avg0022(i_rIput := INT_TO_REAL(A0022), i_uiSmplCnt := fA0022, i_xErrRst := _rt19.Q, q_rOput => Pv12a); // SE_TBX.Filter_MovingAverage

// NETWORK 20
//   A0023: Module_4 : | AT %IW32
//   fA0023: AT %MW119
//   Run: run | AT %M?9
//   gGas: AT %MD28
_rt20(CLK := Run);
avg0023(i_rIput := INT_TO_REAL(A0023), i_uiSmplCnt := fA0023, i_xErrRst := _rt20.Q, q_rOput => gGas); // SE_TBX.Filter_MovingAverage

// NETWORK 21
//   A0024: Module_4 : | AT %IW33
//   fA0024: AT %MW120
//   Run: run | AT %M?9
//   gTerm: AT %MD49
_rt21(CLK := Run);
avg0024(i_rIput := INT_TO_REAL(A0024), i_uiSmplCnt := fA0024, i_xErrRst := _rt21.Q, q_rOput => gTerm); // SE_TBX.Filter_MovingAverage

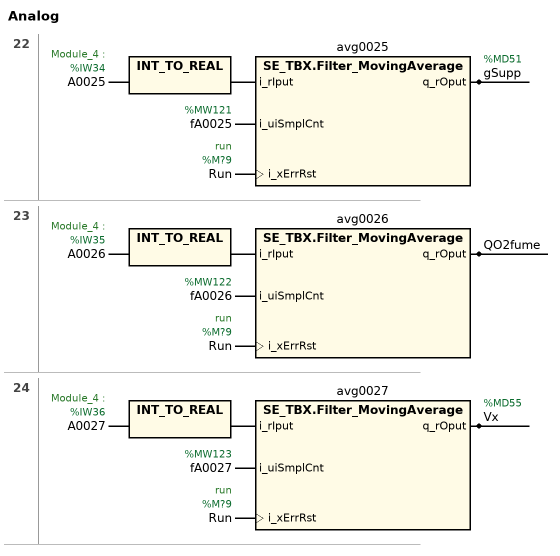
// NETWORK 22
//   A0025: Module_4 : | AT %IW34
//   fA0025: AT %MW121
//   Run: run | AT %M?9
//   gSupp: AT %MD51
_rt22(CLK := Run);
avg0025(i_rIput := INT_TO_REAL(A0025), i_uiSmplCnt := fA0025, i_xErrRst := _rt22.Q, q_rOput => gSupp); // SE_TBX.Filter_MovingAverage

// NETWORK 23
//   A0026: Module_4 : | AT %IW35
//   fA0026: AT %MW122
//   Run: run | AT %M?9
_rt23(CLK := Run);
avg0026(i_rIput := INT_TO_REAL(A0026), i_uiSmplCnt := fA0026, i_xErrRst := _rt23.Q, q_rOput => QO2fume); // SE_TBX.Filter_MovingAverage

// NETWORK 24
//   A0027: Module_4 : | AT %IW36
//   fA0027: AT %MW123
//   Run: run | AT %M?9
//   Vx: AT %MD55
_rt24(CLK := Run);
avg0027(i_rIput := INT_TO_REAL(A0027), i_uiSmplCnt := fA0027, i_xErrRst := _rt24.Q, q_rOput => Vx); // SE_TBX.Filter_MovingAverage

END_PROGRAM

// MyController/Application/HiddenPOU
FUNCTION HiddenPOU : BOOL

VAR_INPUT
	pHiddenFunc: POINTER TO WORD;
END_VAR
VAR
	pRead: POINTER TO BYTE;
	pWrite: POINTER TO BYTE;
END_VAR

pRead := pHiddenFunc + 400;
pWrite := pHiddenFunc + 4400;
HiddenPOU := TRUE;

END_FUNCTION

// MyController/Application/Prog/SafeTmr
PROGRAM SafeTmr
VAR
	tonMeo1: TON;
	rsMeo1: RS;

	tonMeo2: TON;
	rsMeo2: RS;
	tonMeo3: TON;
	rsMeo3: RS;

	tonAl1: TON;
	rsAl1: RS;
END_VAR
VAR // added by the converter: edge detectors and wires of the graphical bodies
    _rt1, _rt2 : R_TRIG;
END_VAR

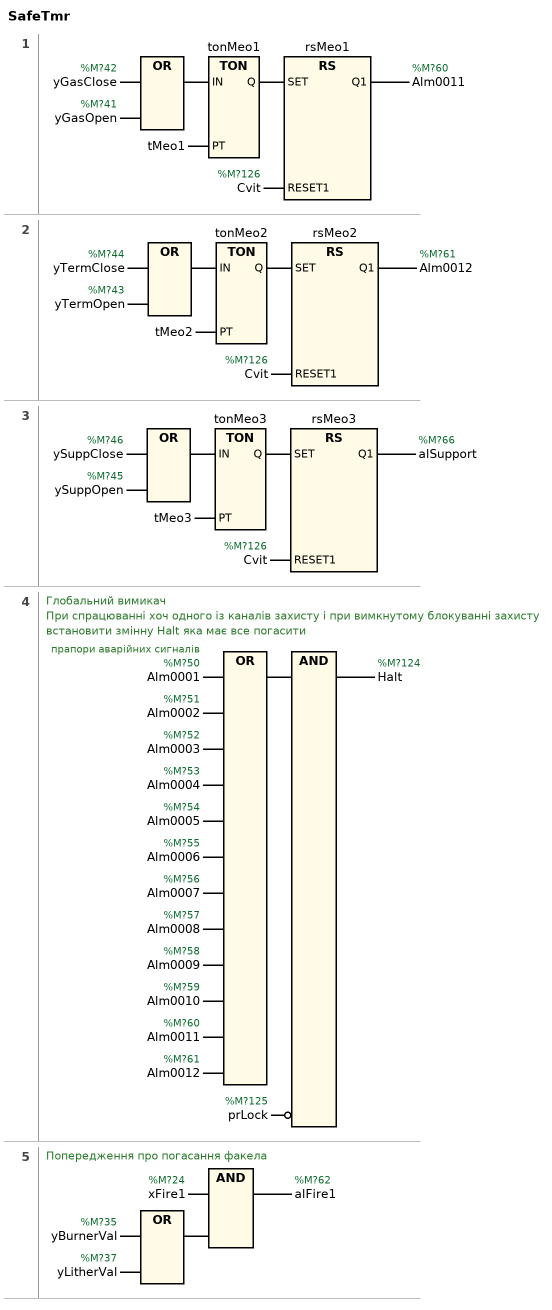
// NETWORK 1
//   yGasClose: AT %M?42
//   yGasOpen: AT %M?41
//   Cvit: AT %M?126
//   Alm0011: AT %M?60
tonMeo1(IN := yGasClose OR yGasOpen, PT := tMeo1); // TON
rsMeo1(SET := tonMeo1.Q, RESET1 := Cvit); // RS
Alm0011 := rsMeo1.Q1;

// NETWORK 2
//   yTermClose: AT %M?44
//   yTermOpen: AT %M?43
//   Cvit: AT %M?126
//   Alm0012: AT %M?61
tonMeo2(IN := yTermClose OR yTermOpen, PT := tMeo2); // TON
rsMeo2(SET := tonMeo2.Q, RESET1 := Cvit); // RS
Alm0012 := rsMeo2.Q1;

// NETWORK 3
//   ySuppClose: AT %M?46
//   ySuppOpen: AT %M?45
//   Cvit: AT %M?126
//   alSupport: AT %M?66
tonMeo3(IN := ySuppClose OR ySuppOpen, PT := tMeo3); // TON
rsMeo3(SET := tonMeo3.Q, RESET1 := Cvit); // RS
alSupport := rsMeo3.Q1;

// NETWORK 4
// Глобальний вимикач
// При спрацюванні хоч одного із каналів захисту і при вимкнутому блокуванні захисту
// встановити змінну Halt яка має все погасити
//   Alm0001: прапори аварійних сигналів | AT %M?50
//   Alm0002: AT %M?51
//   Alm0003: AT %M?52
//   Alm0004: AT %M?53
//   Alm0005: AT %M?54
//   Alm0006: AT %M?55
//   Alm0007: AT %M?56
//   Alm0008: AT %M?57
//   Alm0009: AT %M?58
//   Alm0010: AT %M?59
//   Alm0011: AT %M?60
//   Alm0012: AT %M?61
//   prLock: AT %M?125
//   Halt: AT %M?124
Halt := (Alm0001 OR Alm0002 OR Alm0003 OR Alm0004 OR Alm0005 OR Alm0006 OR Alm0007 OR Alm0008 OR Alm0009 OR Alm0010 OR Alm0011 OR Alm0012) AND NOT prLock;

// NETWORK 5
// Попередження про погасання факела
//   xFire1: AT %M?24
//   yBurnerVal: AT %M?35
//   yLitherVal: AT %M?37
//   alFire1: AT %M?62
alFire1 := xFire1 AND (yBurnerVal OR yLitherVal);

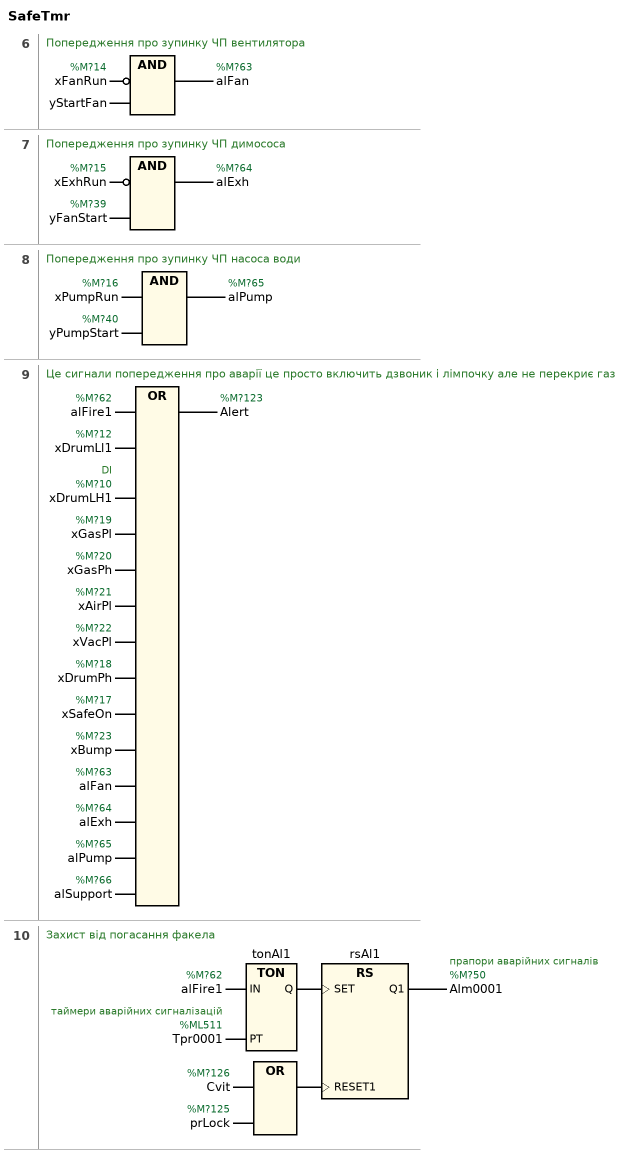
// NETWORK 6
// Попередження про зупинку ЧП вентилятора
//   xFanRun: AT %M?14
//   alFan: AT %M?63
alFan := NOT xFanRun AND yStartFan;

// NETWORK 7
// Попередження про зупинку ЧП димососа
//   xExhRun: AT %M?15
//   yFanStart: AT %M?39
//   alExh: AT %M?64
alExh := NOT xExhRun AND yFanStart;

// NETWORK 8
// Попередження про зупинку ЧП насоса води
//   xPumpRun: AT %M?16
//   yPumpStart: AT %M?40
//   alPump: AT %M?65
alPump := xPumpRun AND yPumpStart;

// NETWORK 9
// Це сигнали попередження про аварії це просто включить дзвоник і лімпочку але не перекриє газ
//   alFire1: AT %M?62
//   xDrumLl1: AT %M?12
//   xDrumLH1: DI | AT %M?10
//   xGasPl: AT %M?19
//   xGasPh: AT %M?20
//   xAirPl: AT %M?21
//   xVacPl: AT %M?22
//   xDrumPh: AT %M?18
//   xSafeOn: AT %M?17
//   xBump: AT %M?23
//   alFan: AT %M?63
//   alExh: AT %M?64
//   alPump: AT %M?65
//   alSupport: AT %M?66
//   Alert: AT %M?123
Alert := alFire1 OR xDrumLl1 OR xDrumLH1 OR xGasPl OR xGasPh OR xAirPl OR xVacPl OR xDrumPh OR xSafeOn OR xBump OR alFan OR alExh OR alPump OR alSupport;

// NETWORK 10
// Захист від погасання факела
//   alFire1: AT %M?62
//   Tpr0001: таймери аварійних сигналізацій | AT %ML511
//   Cvit: AT %M?126
//   prLock: AT %M?125
//   Alm0001: прапори аварійних сигналів | AT %M?50
tonAl1(IN := alFire1, PT := Tpr0001); // TON
_rt1(CLK := tonAl1.Q);
_rt2(CLK := Cvit OR prLock);
rsAl1(SET := _rt1.Q, RESET1 := _rt2.Q); // RS
Alm0001 := rsAl1.Q1;

END_PROGRAM
